DEVICE_TYPE _TCREST
  (* Standard: 61499-2 *)
  (* Version 0.1, 2017-00-01, hpea485, UOA *)
  RESOURCE c1 : _Core102
  END_RESOURCE
  RESOURCE c2 : _Core102
  END_RESOURCE
  RESOURCE c3 : _Core102
  END_RESOURCE
  RESOURCE c4 : _Core102
  END_RESOURCE
END_DEVICE_TYPE
